// TwinCAT 3 PLC project Untitled1
// ProgramVersion: 3.1.4023.0
// libraries:
//   Tc2_MC2, * (Beckhoff Automation GmbH)
//   Tc2_Standard, * (Beckhoff Automation GmbH)
//   Tc2_System, * (Beckhoff Automation GmbH)
//   Tc2_Utilities, * (Beckhoff Automation GmbH)
//   Tc3_JsonXml, * (Beckhoff Automation GmbH)
//   Tc3_Module, * (Beckhoff Automation GmbH)
// project tree:
//   DUTs/ Bundle.TcDUT (not stored), Interval.TcDUT (not stored), PositionMaterials.TcDUT, SuctionPad.TcDUT (not stored)
//   DUTs/Enums/ A22.TcDUT (not stored), Cardboard.TcDUT (not stored), CornerGuard.TcDUT (not stored), Homing.TcDUT (not stored), SectionEnum.TcDUT (not stored), Surface.TcDUT
//   DUTs/Insertion/Drives/ ClearLinkMC.TcPOU, ServoNC.TcPOU, SimplePiston.TcPOU (not stored), TeknicHW.TcPOU (not stored)
//   DUTs/Insertion/ Insertion.TcPOU (not stored)
//   DUTs/Insertion/ABSTRACT/ FBA_Drive.TcPOU (not stored), I_ContinuousDrive.TcIO (not stored), I_Drive.TcIO (not stored), I_EncodedDrive.TcIO (not stored), I_PositionalDrive.TcIO (not stored)
//   DUTs/Machines/ FoldingMachine.TcPOU (not stored), KukaRobot.TcPOU (not stored), RobotA22.TcPOU, WrapMachine.TcPOU (not stored)
//   DUTs/Material Holders/ MaterialHolder.TcPOU, SkidMagazine.TcPOU (not stored), HmiSlotOccupancy.TcDUT
//   GVLs/ ContainerArrays.TcGVL, GVL.TcGVL (not stored), Hardware.TcGVL
//   / PlcTask.TcTTO (not stored)
//   POUs/A22 - Cardboard-Corner Guard/AOIs/ AOI_LoadCornerGuard.TcPOU, AOI_LoadFlatCardboard.TcPOU
//   POUs/A22 - Cardboard-Corner Guard/ CardboardCornerGuardEx.TcPOU
//   POUs/Hardware Calls/ SuctionQualityPtrArr.TcPOU (not stored), SetSuctionsPtrArr.TcPOU (not stored), CallHardwareModules.TcPOU, SuctionQuality.TcPOU, SetSuctions.TcPOU (not stored), SetupHardware.TcPOU
//   POUs/ MAIN.TcPOU, BundleJsonDemo.TcPOU
//   POUs/Materials/ GetMaterialLength.TcPOU (not stored), GetMaterialLengthFromCode.TcPOU (not stored), GetPairMasterLength.TcPOU (not stored), GetPositionMasterLength.TcPOU (not stored), MatchesMaterialType.TcPOU (not stored)
//   POUs/Utility/ CEILING.TcPOU (not stored), IntegerBitAccess.TcPOU, IntegerToBoolArray.TcPOU, WithinTolerance.TcPOU (not stored)
// real-time tasks:
//   TASK PlcTask: cycle T#10ms, priority 20, ADS port 350
// I/O:
//   DEVICE Device 1 (TC3 EIP Scanner), AmsNetId 5.131.216.41.2.1
//     ClearLink // <INFO> 169.254.0.152, ClearLink (ProdCode: 1, Rev: 2.93, Mac: 24:15:10:b0:30:37) </INFO> <EDS> C:\TwinCAT\3.1\Config\Io\EtherNetIP\clearlink_2.92.eds </EDS>

// ---- DUTs/Enums/Surface.TcDUT
{attribute 'qualified_only'}
//{attribute 'strict'}
TYPE Surface :
(
	TOP,
	LEFT,
	RIGHT,
	BOTTOM,
	
	TOP_LEFT,
	TOP_RIGHT,
	BOTTOM_LEFT,
	BOTTOM_RIGHT,
	
	size
);
END_TYPE

// ---- DUTs/Material Holders/HmiSlotOccupancy.TcDUT
TYPE HmiSlotOccupancy :
STRUCT
	material : STRING;
	occupied : BOOL;
END_STRUCT
END_TYPE

// ---- DUTs/PositionMaterials.TcDUT
TYPE PositionMaterials :
STRUCT
	position : REAL; //:= GVL.nullPos; //default value is set to predefined constant if bundle needs less than 32 position material pairs
	
	top : STRING;
	right : STRING;
	left : STRING;
	//sides : STRING;
	bottom : STRING;
	
	topLeft : STRING;
	topLeftFold : USINT;
	
	topRight : STRING;
	topRightFold : USINT;
	
	bottomLeft : STRING;
	bottomLeftFold : USINT;
	
	bottomRight : STRING;
	bottomRightFold : USINT;

	wrapPoints : USINT;
	wrapRotations : USINT;
END_STRUCT
END_TYPE

// ---- GVLs/ContainerArrays.TcGVL
//{attribute 'qualified_only'}
VAR_GLOBAL //data arrays to be passed into material holder FBs - do not access directly
	
	skidSlotsA22Left, skidSlotsA22Right : ARRAY[1..Cardboard.size-1] OF STRING; //cardboard skid
	skidOccupancyA22Left, skidOccupancyA22Right : ARRAY[1...Cardboard.size-1] OF BOOL := [(Cardboard.size-1)(TRUE)];
	skidHmiA22Left, skidHmiA22Right : ARRAY[1...Cardboard.size-1] OF HmiSlotOccupancy;
	
	magazineSlotsA22Left, magazineSlotsA22Right : ARRAY[1..CornerGuard.size-1] OF STRING; //corner guard magazine
	magazineOccupancyA22Left, magazineOccupancyA22Right : ARRAY[1..CornerGuard.size-1] OF BOOL := [(CornerGuard.size-1)(TRUE)];
	magazineHmiA22Left, magazineHmiA22Right : ARRAY[1..CornerGuard.size-1] OF HmiSlotOccupancy;
END_VAR

// ---- GVLs/Hardware.TcGVL
//{attribute 'qualified_only'}
VAR_GLOBAL //complete modules
	robot3, robot4 : RobotA22;
	
	benderA22Left : FoldingMachine;
	
	skidA22Left, skidA22Right : SkidMagazine;
	magazineA22Left, magazineA22Right : SkidMagazine;
	
	wrapperA22 : WrapMachine;
	overhead : STRING;
	
	horizontalDriveA22Left, horizontalDriveA22Right : ServoNC;
	verticalDriveA22Left, verticalDriveA22Right : ClearLinkMC;
	pistonA22Bottom : SimplePiston;
	
	(*
	each of these suction arrays are composed of 3 pads
	pad [2] is the corner pad used for corner guards
	pads [1] and [3] are the outer pads used for corner cardboards
	*)
	suctionA22TopLeft : ARRAY[1..3] OF SuctionPad;
	suctionA22TopRight : ARRAY[1..3] OF SuctionPad;
	suctionA22BottomLeft : ARRAY[1..3] OF SuctionPad; 
	suctionA22BottomRight : ARRAY[1..3] OF SuctionPad;
	
	suctionA22Bottom : SuctionPad;
END_VAR

// ---- DUTs/Machines/RobotA22.TcPOU
FUNCTION_BLOCK RobotA22 EXTENDS KukaRobot
VAR_OUTPUT //from outputs array
	taskID : A22;
	param1 : INT;
	param2 : INT;
	Xmm : INT;
	Ymm : INT;
	Zmm : INT;
	angle : INT;
	foldPosition0 : INT;
	foldPosition1 : INT;
END_VAR
VAR_OUTPUT //from inputs array
	tool : SectionEnum := SectionEnum.CARDBOARD_CORNERGUARD;
	suspendedMaterial : STRING;
	
	completedTask : A22;
	eoatDistance : INT;
	cardboardAvailability : INT;
	cornerGuardAvailability : INT;
	materialAtHoldingPosition : INT;
	//grp6
	//grp7
	
	wrapSafetyIn : BOOL;
	
END_VAR
VAR //HMI data
	reservationEnum : SectionEnum;
	hmiTask : STRING;
	hmiTool : STRING;
END_VAR

{warning disable C0195}
SUPER^();

outputs[1] := taskID;
outputs[2] := param1;
outputs[3] := param2;
outputs[4] := Xmm;
outputs[5] := Ymm;
outputs[6] := Zmm;
outputs[7] := angle;
outputs[8] := foldPosition0;
outputs[9] := foldPosition1;

refreshParameters();

reservationEnum := reservation;
IF reservationEnum = SectionEnum.NULL_SECTION THEN
	hmiReservation := 'N/A';
ELSE
	hmiReservation := TO_STRING(reservationEnum);
END_IF

hmiTask := TO_STRING(taskID);
hmiTool := TO_STRING(tool);

{attribute 'monitoring' := 'call'}
PROPERTY Busy : BOOL
GET
VAR
	//emptyOutput : ARRAY[1..50] OF INT;
END_VAR
//Busy stays TRUE until outputs are cleared AND completed task has elapsed
//Ready is always inverse of Busy
refreshParameters();

Busy := taskID <> 0 OR completedTask <> 0;
END_GET
END_PROPERTY

METHOD clearCommand : BOOL
VAR_INPUT
END_VAR
SUPER^.clearCommand();

refreshParameters();
END_METHOD

{attribute 'monitoring' := 'call'}
PROPERTY Done : BOOL
GET
refreshParameters();

Done :=
	completedTask = taskID AND
	taskID <> 0 AND
	completedTask <> 0;
END_GET
END_PROPERTY

{attribute 'monitoring' := 'call'}
PROPERTY HoldMaterial : STRING
GET
HoldMaterial := suspendedMaterial;
END_GET
SET
suspendedMaterial := HoldMaterial;
END_SET
END_PROPERTY

{attribute 'monitoring' := 'call'}
PROPERTY Ready : BOOL
GET
refreshParameters();

Ready := taskID = 0 AND completedTask = 0;
END_GET
END_PROPERTY

METHOD PRIVATE refreshParameters : BOOL
VAR_INPUT
END_VAR
{warning disable C0196}
taskID := outputs[1];
param1 := outputs[2];
param2 := outputs[3];
Xmm := outputs[4];
Ymm := outputs[5];
Zmm := outputs[6];
angle := outputs[7];
foldPosition0 := outputs[8];
foldPosition1 := outputs[9];

completedTask := inputs[1];
(*
eoatDistance := inputs[2];
magazineAvailability := inputs[3];
chipboardSkidInPosition := inputs[4];
materialAtHoldingPosition := inputs[5];
//robotEOAT := inputs[6];

strapSafetyIn := inputs[4].15;
*)
END_METHOD

METHOD setGroup : BOOL
VAR_INPUT
	group : INT;
	value : INT;
END_VAR
SUPER^.setGroup(group := group, value := value);

refreshParameters();
END_METHOD

METHOD setParameters : BOOL
VAR_INPUT
	newTaskID : INT;
	newParam1 : INT;
	newParam2 : INT;
	newXmm : INT;
	newYmm : INT;
	newZmm : INT;
	newAngle : INT;
	newStagingOccupancy : INT;
	newInsertionSuctionStatus : INT;
	newMagazineStatus : INT; //unused
	newInspectionValue : INT;
END_VAR
setGroup(group := 1, value := newTaskID);
setGroup(group := 2, value := newParam1);
setGroup(group := 3, value := newParam2);
setGroup(group := 4, value := newXmm);
setGroup(group := 5, value := newYmm);
setGroup(group := 6, value := newZmm);
setGroup(group := 7, value := newAngle);

newStagingOccupancy.15 := NOT wrapperA22.enable AND NOT wrapperA22.execute;
setGroup(group := 8, value := newStagingOccupancy);

setGroup(group := 9, value := newInsertionSuctionStatus);
setGroup(group := 10, value := newMagazineStatus);
setGroup(group := 11, value := newInspectionValue);

refreshParameters();
END_METHOD

END_FUNCTION_BLOCK

// ---- DUTs/Insertion/Drives/ServoNC.TcPOU
FUNCTION_BLOCK ServoNC EXTENDS FBA_Drive IMPLEMENTS I_EncodedDrive
VAR_OUTPUT	
	ready : BOOL;
	position : LREAL;
END_VAR
VAR
	axis : AXIS_REF;
	
	mcReadPosition : MC_ReadActualPosition;
	mcReset : MC_Reset;
	
	mcPower : MC_Power;
	mcMoveAbsolute : MC_MoveAbsolute;
	mcMoveRelative : MC_MoveRelative;
	mcMoveVelocity : MC_MoveVelocity;
	
	mcSetPosition : MC_SetPosition;
	mcStop : MC_Stop;
END_VAR
VAR_STAT CONSTANT
	targetingVelocity : INT := 500;
	continuousVelocity : INT := 200;
END_VAR

IF home OR outerLimit OR innerLimit THEN
	stop();
END_IF

blocks();

mcReset.Execute := FALSE;
mcMoveAbsolute.Execute := FALSE;
mcMoveRelative.Execute := FALSE;
mcMoveVelocity.Execute := FALSE;
mcSetPosition.Execute := FALSE;
mcStop.Execute := FALSE;

blocks();

ready := bEnable AND NOT busy AND homeSet;

METHOD PRIVATE blocks : BOOL
mcReadPosition(
	Axis:= axis, 
	Enable:= TRUE, 
	Valid=> , 
	Busy=> , 
	Error=> , 
	ErrorID=> , 
	Position=> position);

mcReset(
	Axis:= axis, 
	Execute:= , 
	Done=> , 
	Busy=> , 
	Error=> , 
	ErrorID=> );

mcPower(
	Axis:= axis, 
	Enable:= bEnable, 
	Enable_Positive:= TRUE, 
	Enable_Negative:= TRUE, 
	Override:= 100, 
	BufferMode:= , 
	Options:= , 
	Status=> , 
	Busy=> , 
	Active=> , 
	Error=> , 
	ErrorID=> );

mcMoveAbsolute(
	Axis:= axis, 
	Execute:= , 
	Position:= , 
	Velocity:= targetingVelocity, 
	Acceleration:= , 
	Deceleration:= , 
	Jerk:= , 
	BufferMode:= , 
	Options:= , 
	Done=> , 
	Busy=> , 
	Active=> , 
	CommandAborted=> , 
	Error=> , 
	ErrorID=> );
	
mcMoveRelative(
	Axis:= axis, 
	Execute:= , 
	Distance:= ,
	Velocity:= targetingVelocity, 
	Acceleration:= , 
	Deceleration:= , 
	Jerk:= , 
	BufferMode:= , 
	Options:= , 
	Done=> , 
	Busy=> , 
	Active=> , 
	CommandAborted=> , 
	Error=> , 
	ErrorID=> );
	
mcMoveVelocity( //stopped with stop();
	Axis:= axis, 
	Execute:= , 
	Velocity:= continuousVelocity, 
	Acceleration:= , 
	Deceleration:= , 
	Jerk:= , 
	Direction:= , 
	BufferMode:= , 
	Options:= , 
	InVelocity=> , 
	Busy=> , 
	Active=> , 
	CommandAborted=> , 
	Error=> , 
	ErrorID=> );
	
mcSetPosition(
	Axis:= axis, 
	Execute:= , 
	Position:= , 
	Mode:= , 
	Options:= , 
	Done=> , 
	Busy=> , 
	Error=> , 
	ErrorID=> );
	
mcStop(
	Axis:= axis, 
	Execute:= , 
	Deceleration:= , 
	Jerk:= , 
	Options:= , 
	Done=> , 
	Busy=> , 
	Active=> , 
	CommandAborted=> , 
	Error=> , 
	ErrorID=> );
END_METHOD

PROPERTY Busy : BOOL
GET
busy := 
	mcMoveAbsolute.Busy OR 
	mcMoveRelative.Busy OR 
	mcMoveVelocity.Busy OR 
	mcSetPosition.Busy OR 
	mcReset.Busy OR 
	mcStop.Busy OR 
	step <> 0;
END_GET
END_PROPERTY

PROPERTY CurrentPosition : LREAL
GET
CurrentPosition := position;
END_GET
SET
position := CurrentPosition;
END_SET
END_PROPERTY

PROPERTY Error : BOOL
GET
error := 
	mcMoveAbsolute.Error OR 
	mcMoveRelative.Error OR 
	mcMoveVelocity.Error OR 
	mcSetPosition.Error OR 
	mcReset.Error OR 
	mcStop.Error;
END_GET
END_PROPERTY

METHOD homingSequence : BOOL
CASE step OF
	Homing.IDLE:
		IF bEnable THEN
			step := Homing.IN;
		END_IF
		
	Homing.IN:
		IF mcMoveVelocity.Execute AND NOT innerLimit THEN
			mcMoveVelocity.Execute := FALSE;
			step := Homing.OUT;
			RETURN;
		END_IF
		
		mcMoveVelocity.Direction := MC_Negative_Direction;
		mcMoveVelocity.Execute := TRUE;
		
	Homing.OUT:
		IF mcMoveVelocity.Execute AND NOT home THEN //if reached home
			mcMoveVelocity.Execute := FALSE;
			step := Homing.STOP;
			RETURN;
		END_IF
		
		mcMoveVelocity.Direction := MC_Positive_Direction;
		mcMoveVelocity.Execute := TRUE;
		
	Homing.STOP:
		IF mcStop.Execute AND mcStop.Done THEN
			mcStop.Execute := FALSE;
			step := Homing.SET;
			RETURN;
		END_IF
		
		mcStop.Execute := TRUE;
		
	Homing.SET:
		IF mcSetPosition.Execute AND mcSetPosition.Done THEN
			mcSetPosition.Execute := FALSE;
			homingSequence := TRUE;
			step := Homing.IDLE;
			RETURN;
		END_IF
		
		mcSetPosition.Position := 0;
		mcSetPosition.Execute := TRUE;
		
END_CASE
END_METHOD

METHOD moveAbsolute : BOOL
VAR_INPUT
	newTarget : LREAL;
END_VAR
(*
VAR_OUTPUT
	fault : BOOL;
END_VAR
*)
IF NOT busy AND NOT error THEN
	mcMoveAbsolute.Position := newTarget;
	mcMoveAbsolute.Execute := TRUE;
END_IF

moveAbsolute := (*mcMoveAbsolute.Done AND mcMoveAbsolute.Active;*)
	position = newTarget;
END_METHOD

METHOD moveContinuous : BOOL
VAR_INPUT
	//direction : BOOL; //direction (F = inwards, T = outwards)
	direction : MC_Direction;
END_VAR
(*
IF mcMoveVelocity.Active THEN
	stop();
END_IF

IF NOT mcStop.Done THEN
	RETURN;
END_IF
*)
(*
IF direction THEN
	mcMoveVelocity.Direction := MC_Positive_Direction;
ELSE
	mcMoveVelocity.Direction := MC_Negative_Direction;
END_IF
*)
mcMoveVelocity.Direction := direction;

IF NOT mcMoveVelocity.Error THEN
	mcMoveVelocity.Execute := TRUE;
	moveContinuous := TRUE;
END_IF
END_METHOD

METHOD moveRelative : BOOL
VAR_INPUT
	distance : LREAL;
END_VAR
mcMoveRelative.Distance := distance;

moveRelative := mcMoveRelative.Done;
END_METHOD

METHOD reset : BOOL
VAR_INPUT
END_VAR
mcReset.Execute := TRUE;

reset := mcReset.Done;
END_METHOD

METHOD stop : BOOL
VAR_INPUT
END_VAR
mcStop.Execute := TRUE;
END_METHOD

PROPERTY TargetPosition : LREAL
GET
END_GET
SET
moveAbsolute(newTarget := TargetPosition);
END_SET
END_PROPERTY

END_FUNCTION_BLOCK

// ---- DUTs/Insertion/Drives/ClearLinkMC.TcPOU
FUNCTION_BLOCK ClearLinkMC EXTENDS FBA_Drive IMPLEMENTS I_EncodedDrive //I_PositionalDrive, I_ContinuousDrive
VAR_OUTPUT
	pulse AT %Q* : INT; //num pulses
	outputRegister AT %Q* : INT;
	brakeRelease AT %Q* : BOOL;
	
	A : BOOL; //direction (F = inwards, T = outwards)
	B : BOOL; //home bit
	clear : BOOL;
	
	hlfb AT %I* : REAL; //high level feedback, if -9999 then servo is idle
	position, targetPos : LREAL;
END_VAR
VAR
	pulseRequest : INT;
	
	minHoming : TON;
	resetTimer : TP;
	
	mode : (DISABLE, HOLD, TARGET, CONTINUOUS, RESET_ERR);
END_VAR
VAR_STAT CONSTANT
	resetTime : TIME := T#1000MS;
	unitsPerPulse : INT := 800; //800 Teknic units per revolution
	distancePerPulse : INT := 5; //5mm per revolution
END_VAR

//M-connector output register
outputRegister.0 := bEnable; 	//enable
outputRegister.1 := A; 			//direction bit
outputRegister.2 := B; 			//homing bit - set to TRUE after startup to begin homing, then set to FALSE to finish homing
outputRegister.3 := clear; 		//reset bit

resetTimer(IN:= , PT:= resetTime, Q=> clear, ET=> ); //reset timer

IF NOT bEnable THEN
	homingComplete := FALSE;
	mode := HOLD;
END_IF

override(); //if sensor limits are reached, this method blocks motion that would exceed the limits

CASE mode OF		
	HOLD: //hold current position, no motion
		pulse := 0;
		pulseRequest := 0;
	
	TARGET:	//target a given position
		IF WithinTolerance(position, targetPos, distancePerPulse) THEN
			pulseRequest := 0;
			mode := HOLD;
			
		ELSIF NOT Busy THEN
			A :=  position < targetPos;
			(*
			2 options to traverse to a target position:
				a)  send all pulses at once - single continuous motion but may exceed limits
				b)  1 pulse at a time - choppy but safer
			*)
			//pulseRequest := TO_INT(ABS(position - targetPos)/distancePerPulse);
			pulseRequest := 1;
			
		END_IF
		
	CONTINUOUS: //single pulses in the direction specified by moveContinuous()
		pulseRequest := 1;
		
	RESET_ERR: //reset pulse, servo may need to be rehomed aftewards
		pulse := 0;
		pulseRequest := 0;
		resetTimer.IN := TRUE;
		
		IF resetTimer.Q THEN
			resetTimer.IN := FALSE;
			mode := HOLD;
		END_IF
		
END_CASE

sequence();

PROPERTY Busy : BOOL
GET
Busy := hlfb <> -9999;
END_GET
END_PROPERTY

PROPERTY CurrentPosition : LREAL
GET
CurrentPosition := position;
END_GET
SET
position := CurrentPosition;
END_SET
END_PROPERTY

PROPERTY Error : BOOL
GET
END_GET
END_PROPERTY

METHOD homingSequence : BOOL
minHoming(IN:= , PT:= T#1S, Q=> , ET=> ); //IN and OUT should be held for at least 1 second - may be removed for deployment

IF NOT bEnable THEN //homing does not begin until software enable
	RETURN;
END_IF

CASE step OF
	Homing.IDLE:
		bEnable := FALSE;
		A := FALSE;
		B := FALSE;
		brakeRelease := TRUE;
		
		homingComplete := FALSE;
		step := Homing.IN;
		
	Homing.IN: //let insertion drop to inner limit before homing
		bEnable := FALSE;
		A := FALSE;
		B := FALSE;
		brakeRelease := TRUE;
		
		minHoming.IN := TRUE;
		
		IF NOT innerLimit AND minHoming.Q THEN
			minHoming.IN := FALSE;
			step := Homing.OUT;
		END_IF
	
	Homing.OUT:
		bEnable := TRUE;
		A := FALSE;
		B := TRUE;
		brakeRelease := TRUE;
		
		minHoming.IN := TRUE;
		
		IF NOT home AND minHoming.Q THEN
			minHoming.IN := FALSE;
			step := Homing.DONE;
		END_IF
		
	Homing.DONE:
		bEnable := TRUE;
		A := FALSE;
		B := FALSE;
		brakeRelease := TRUE;
			
		position := 0;
		
		homingComplete := TRUE;
		homingSequence := TRUE;
		
		mode := HOLD;
		step := Homing.IDLE;
	
END_CASE
END_METHOD

METHOD moveAbsolute : BOOL
VAR_INPUT
	newTarget : LREAL;
END_VAR
targetPos := newTarget;
mode := TARGET;
END_METHOD

METHOD moveContinuous : BOOL
VAR_INPUT
	direction : MC_Direction;
END_VAR
IF direction = MC_Negative_Direction THEN
	A := FALSE;
ELSIF direction = MC_Positive_Direction THEN
	A := TRUE;
END_IF

mode := CONTINUOUS;
END_METHOD

METHOD moveRelative : BOOL
VAR_INPUT
	distance : LREAL;
END_VAR
targetPos := targetPos + distance;

mode := TARGET;
END_METHOD

METHOD PRIVATE override : BOOL
VAR_INPUT
END_VAR
(*
IF (*NOT*) home THEN //block outwards motion
	position := 0;
	IF A THEN
		mode := HOLD;
	END_IF
	
ELSIF (*NOT*) outerLimit AND_THEN A THEN //block outwards motion
	mode := HOLD;

ELSIF (*NOT*) innerLimit AND_THEN NOT A THEN //block inwards motion
	mode := HOLD;
	
END_IF
*)


IF
	((*NOT*) home AND_THEN A) OR
	((*NOT*) outerLimit AND_THEN A) OR
	((*NOT*) innerLimit AND_THEN NOT A)
THEN
	mode := HOLD;
END_IF


IF (*NOT*) home THEN //block outwards motion
	position := 0;
END_IF
END_METHOD

METHOD reset : BOOL
VAR_INPUT
END_VAR
mode := RESET_ERR;
END_METHOD

METHOD PRIVATE sequence : BOOL
VAR_INPUT
END_VAR
IF Busy THEN //servo is active
	IF A THEN //positive direction
		position := position + (distancePerPulse * pulse);
	ELSE //negative direction
		position := position - (distancePerPulse * pulse);
	END_IF
	pulse := 0; //pulses already received, can be set to 0 so position change is not compounded

ELSIF pulse = 0 THEN //servo is not active
	pulse := pulseRequest;
	pulseRequest := 0; //remove this if not working as intended
	
END_IF
END_METHOD

METHOD stop : BOOL
VAR_INPUT
END_VAR
mode := HOLD;
END_METHOD

PROPERTY TargetPosition : LREAL
GET
END_GET
SET
targetPos := TargetPosition;
END_SET
END_PROPERTY

END_FUNCTION_BLOCK

// ---- DUTs/Material Holders/MaterialHolder.TcPOU
FUNCTION_BLOCK MaterialHolder
VAR_IN_OUT
	slots : ARRAY[*] OF STRING;
	occupied : ARRAY[*] OF BOOL;
	
	hmiTable : ARRAY[*] OF HmiSlotOccupancy;
END_VAR

IF hmiTable <> 0 THEN
	writeHmiTable();
END_IF

METHOD clear : BOOL
VAR_INPUT
END_VAR
MEMSET(ADR(slots), 0, SIZEOF(slots));
END_METHOD

METHOD findSlot : BOOL
VAR_INPUT
	materialID : STRING;
END_VAR
VAR_OUTPUT
	index : INT := 0;
END_VAR
VAR
	i : DINT;
END_VAR
IF materialID = '' THEN
	RETURN;
END_IF

FOR i:=LOWER_BOUND(slots, 1) TO UPPER_BOUND(slots, 1) BY 1 DO
	IF slots[i] = materialID THEN
		index := TO_INT(i);
		findSlot := TRUE;
		RETURN;
	END_IF
END_FOR
END_METHOD

METHOD getSlot : STRING
VAR_INPUT
	i : DINT;
END_VAR
VAR_OUTPUT
	error : BOOL;
END_VAR
error := i < LOWER_BOUND(slots, 1) OR i > UPPER_BOUND(slots, 1);

IF error THEN
	RETURN;
END_IF

getSlot := slots[i];
END_METHOD

METHOD getSlotsAsArray : POINTER TO STRING
getSlotsAsArray := ADR(slots);
END_METHOD

METHOD isOccupied : BOOL
VAR_INPUT
	i : DINT;
END_VAR
VAR_OUTPUT
	errorBounds : BOOL;
END_VAR
errorBounds := i < LOWER_BOUND(slots, 1) OR i > UPPER_BOUND(slots, 1);

IF errorBounds THEN
	RETURN;
END_IF

isOccupied := occupied[i];
END_METHOD

METHOD setSlot : BOOL
VAR_INPUT
	i : INT;
	material : STRING;
END_VAR
VAR_OUTPUT
	error : BOOL;
END_VAR
IF i < LOWER_BOUND(slots, 1) OR i > UPPER_BOUND(slots, 1) THEN
	error := TRUE;
	RETURN;
END_IF

slots[i] := material;

IF hmiTable <> 0 THEN
	writeHmiTable();
END_IF
END_METHOD

METHOD PRIVATE writeHmiTable : BOOL
VAR
	i : DINT;
END_VAR
FOR i:=LOWER_BOUND(hmiTable, 1) TO UPPER_BOUND(hmiTable, 1) BY 1 DO
	hmiTable[i].material := slots[i];
	hmiTable[i].occupied := occupied[i];
END_FOR
END_METHOD

END_FUNCTION_BLOCK

// ---- POUs/A22 - Cardboard-Corner Guard/AOIs/AOI_LoadCornerGuard.TcPOU
FUNCTION_BLOCK AOI_LoadCornerGuard
VAR_INPUT
	execute : BOOL;
END_VAR
VAR_IN_OUT CONSTANT
	sectionID : SectionEnum;
END_VAR
VAR_IN_OUT
	robot : RobotA22;
	magazine : SkidMagazine;
	loadedMaterials : ARRAY[*] OF STRING;
END_VAR
VAR_INPUT
	surfaceID : Surface;
	material : STRING;
	
	suctions : POINTER TO SuctionPad; //access from 0 to numPads-1, not LOWER_BOUND to UPPER_BOUND
	numPads : DINT;
END_VAR
VAR_OUTPUT
	donePulse : BOOL; //this signal turns on 1 cycle after done turns true, should not affect the program structure
	done : BOOL;
	busy : BOOL;
	error : BOOL;
	
	recovery : BOOL;
	failCounter : INT;
END_VAR
VAR
	run : BOOL;
	trigger : R_TRIG;
	doneTrigger : R_TRIG;
	
	slot : INT;
	
	suctionTimer : TON;
	step : (IDLE, PREP_ROBOT, GET_FROM_STORAGE, LOAD_TO_INSERTION, COMPLETE, RECOVERY_IDLE, RECOVERY_REMOVE, RECOVERY_LOAD);
	
	i : DINT;
END_VAR
VAR CONSTANT
	suctionDelay : TIME := T#2S;
	suctionDistance : INT := 10;
END_VAR

{warning disable C0371}

trigger(CLK:= execute, Q=> );
doneTrigger(CLK:= done, Q=> donePulse);
busy := trigger.Q OR step > 0;

IF step > IDLE AND_THEN NOT preExecution() THEN //conditions to track before execution
	RETURN;
END_IF

(*
if required bunk was not found on table - restage entire table
if bunk was not loaded correctly - remove bunk, then restage entire table
*)
CASE step OF
	IDLE:
		IF trigger.Q THEN
			recovery := FALSE;
			done := FALSE;
			error := FALSE;
			step := PREP_ROBOT;
		END_IF
		
	PREP_ROBOT:
		robot.clearCommand();
		IF robot.Ready THEN
			step := GET_FROM_STORAGE;
			slot := 0;
		END_IF
		
	GET_FROM_STORAGE:		
		IF NOT magazine.findSlot(materialID := material, index => slot) THEN
			error := TRUE;
			RETURN;
		END_IF
		
		IF robot.eoatDistance < suctionDistance THEN //move from table to robot gripper
			robot.HoldMaterial := magazine.getSlot(i := slot, error => );
		END_IF
		
		IF robot.Done THEN
			step := COMPLETE;
			RETURN;
		ELSIF robot.materialAtHoldingPosition > 0 THEN
			step := LOAD_TO_INSERTION;
			RETURN;
		END_IF
		
		CASE surfaceID OF
			Surface.TOP_LEFT, Surface.TOP_RIGHT:			robot.setGroup(group := 1, value := A22.LOAD_CORNER_GUARD_UPPER);
			Surface.BOTTOM_LEFT, SURFACE.BOTTOM_RIGHT:		robot.setGroup(group := 1, value := A22.LOAD_CORNER_GUARD_LOWER);
		END_CASE
		robot.setGroup(group := 2, value := slot); 
			
	LOAD_TO_INSERTION:
		IF robot.materialAtHoldingPosition > 0 AND robot.HoldMaterial <> '' THEN //move from gripper to insertion
			loadedMaterials[surfaceID] := robot.HoldMaterial;
			robot.HoldMaterial := '';
		END_IF
		
		//numPads/3 <= i < numPads/3 * 2
		FOR i:=(numPads/3)*1 TO (numPads/3)*2-1 BY 1 DO //middle third suctions only
			suctions[i].enable := TRUE;
		END_FOR
		
		IF robot.Done THEN
			suctionTimer.IN := FALSE;
			step := COMPLETE;
			RETURN;
		END_IF
		
		suctionTimer(IN:= , PT:= suctionDelay, Q=> , ET=> );
		suctionTimer.IN := TRUE;
		
		IF suctionTimer.Q THEN
			robot.setGroup(group := 10, value := robot.materialAtHoldingPosition);
		END_IF
	
	COMPLETE:
		robot.clearCommand();
		
		IF //check insertion quality
			SuctionQualityPtrArr(
				suctions := suctions, 
				numPads := numPads, 
				insertionMaterial := loadedMaterials[surfaceID], 
				recipeMaterial := material)
		THEN
			done := TRUE;
			slot := 0;
			step := 0;
			
		ELSE //recovery - remove and reload
			failCounter := failCounter + 1;
			step := RECOVERY_IDLE;
		END_IF
		
		
	//---------RECOVERY-----------------------------------------
	RECOVERY_IDLE:
		robot.clearCommand();
		IF robot.Ready THEN
			step := RECOVERY_REMOVE;
		END_IF
		
	RECOVERY_REMOVE:
		IF robot.Done THEN
			step := RECOVERY_LOAD;
			RETURN;
		END_IF
		
		CASE surfaceID OF
			Surface.TOP_LEFT, Surface.TOP_RIGHT:			robot.setGroup(group := 1, value := A22.REMOVE_CORNER_GUARD_UPPER);
			Surface.BOTTOM_LEFT, SURFACE.BOTTOM_RIGHT:		robot.setGroup(group := 1, value := A22.REMOVE_CORNER_GUARD_LOWER);
		END_CASE
		
	RECOVERY_LOAD:	
		recovery := TRUE;
		error := TRUE;
		
END_CASE

METHOD PRIVATE preExecution : BOOL
VAR_INPUT
END_VAR
{warning disable C0371}
IF material = '' THEN
	done := TRUE;
	RETURN;
END_IF

IF //robot must be ready before execution
	robot.error OR 
	robot.reservation <> sectionID OR 
	robot.tool <> sectionID
THEN
	error := TRUE;
	RETURN;
END_IF

preExecution := TRUE;
END_METHOD

METHOD reset : BOOL
VAR_INPUT
END_VAR
done := FALSE;
error := FALSE;
recovery := FALSE;
slot := 0;
step := 0;

failCounter := 0;
END_METHOD

END_FUNCTION_BLOCK

// ---- POUs/A22 - Cardboard-Corner Guard/AOIs/AOI_LoadFlatCardboard.TcPOU
FUNCTION_BLOCK AOI_LoadFlatCardboard
VAR_INPUT
	execute : BOOL;
END_VAR
VAR_IN_OUT CONSTANT
	sectionID : SectionEnum;
END_VAR
VAR_IN_OUT
	robot : RobotA22;
	skid : SkidMagazine;
	loadedMaterials : ARRAY[*] OF STRING;
END_VAR
VAR_INPUT
	surfaceID : Surface;
	material : STRING;
	
	suctions : POINTER TO SuctionPad; //access from 0 to numPads-1, not LOWER_BOUND to UPPER_BOUND
	numPads : DINT;
END_VAR
VAR_OUTPUT
	donePulse : BOOL;
	done : BOOL;
	busy : BOOL;
	error : BOOL;
	
	recovery : BOOL;
	failCounter : INT;
END_VAR
VAR
	run : BOOL;
	trigger : R_TRIG;
	doneTrigger : R_TRIG;
	
	slot : INT;
	
	suctionTimer : TON;
	step : (IDLE, PREP_ROBOT, GET_FROM_STORAGE, LOAD_TO_INSERTION, COMPLETE, RECOVERY_IDLE, RECOVERY_REMOVE, RECOVERY_WAIT, RECOVERY_LOAD);
	
	i : DINT;
END_VAR
VAR_STAT CONSTANT
	suctionDelay : TIME := T#2S;
	suctionDistance : INT := 10;
END_VAR

{warning disable C0371}

trigger(CLK:= execute, Q=> );
doneTrigger(CLK:= done, Q=> donePulse);
busy := trigger.Q OR step > 0;

IF step > IDLE AND_THEN NOT preExecution() THEN //conditions to track before execution
	RETURN;
END_IF

(*
if bunk was not loaded correctly - remove bunk, then restage entire table
*)
CASE step OF
	IDLE:
		IF trigger.Q THEN
			recovery := FALSE;
			done := FALSE;
			error := FALSE;
			step := PREP_ROBOT;
		END_IF
		
	PREP_ROBOT:
		robot.clearCommand();
		IF robot.Ready THEN
			step := GET_FROM_STORAGE;
			slot := 0;
		END_IF
		
	GET_FROM_STORAGE:		
		IF NOT skid.findSlot(materialID := material, index => slot) THEN
			error := TRUE;
			RETURN;
		END_IF
		
		IF robot.eoatDistance < suctionDistance THEN//move from table to robot gripper
			robot.HoldMaterial := skid.getSlot(i := slot, error => );;
		END_IF
		
		IF robot.Done THEN
			step := COMPLETE;
			RETURN;
		ELSIF robot.materialAtHoldingPosition >= 1 AND robot.materialAtHoldingPosition <= 8 THEN
			step := LOAD_TO_INSERTION;
			RETURN;
		END_IF
		
		CASE surfaceID OF
			Surface.TOP_LEFT, Surface.TOP_RIGHT:			robot.setGroup(group := 1, value := A22.LOAD_CORNER_GUARD_UPPER);
			Surface.BOTTOM_LEFT, SURFACE.BOTTOM_RIGHT:		robot.setGroup(group := 1, value := A22.LOAD_CORNER_GUARD_LOWER);
		END_CASE
		robot.setGroup(group := 2, value := slot); 
			
	LOAD_TO_INSERTION:
		IF robot.materialAtHoldingPosition > 0 AND robot.HoldMaterial <> '' THEN //move from gripper to insertion
			loadedMaterials[surfaceID] := robot.HoldMaterial;
			robot.HoldMaterial := '';
		END_IF
		
		//only bottom cardboard uses suction
		CASE surfaceID OF
			Surface.BOTTOM:		SetSuctionsPtrArr(suctions := suctions, numPads := numPads, state := TRUE);
		END_CASE
		
		IF robot.Done THEN
			suctionTimer.IN := FALSE;
			step := COMPLETE;
			RETURN;
		END_IF
		
		suctionTimer(IN:= , PT:= suctionDelay, Q=> , ET=> );
		suctionTimer.IN := TRUE;
		
		IF suctionTimer.Q THEN
			robot.setGroup(group := 10, value := robot.materialAtHoldingPosition);
		END_IF
	
	COMPLETE:
		robot.clearCommand();
		
		IF //if bottom then check insertion, otherwise done
			surfaceID <> Surface.BOTTOM OR_ELSE 
			SuctionQualityPtrArr(
				suctions := suctions, 
				numPads := numPads, 
				insertionMaterial := loadedMaterials[surfaceID], 
				recipeMaterial := material)
		THEN
			done := TRUE;
			slot := 0;
			step := 0;
			
		ELSE //recovery - remove and reload
			failCounter := failCounter + 1;
			step := RECOVERY_IDLE;
		END_IF
		
	//---------RECOVERY-----------------------------------------
	RECOVERY_IDLE:
		robot.clearCommand();
		IF robot.Ready THEN
			step := RECOVERY_REMOVE;
		END_IF
		
	RECOVERY_REMOVE:
		IF robot.Done THEN
			step := RECOVERY_LOAD;
			RETURN;
		END_IF
		
		CASE surfaceID OF
			Surface.BOTTOM:		robot.setGroup(group := 1, value := A22.REMOVE_CARDBOARD_BOTTOM);
		END_CASE
		
	RECOVERY_LOAD:	
		recovery := TRUE;
		error := TRUE;
		
END_CASE

METHOD PRIVATE preExecution : BOOL
VAR_INPUT
END_VAR
{warning disable C0371}
IF material = '' THEN
	done := TRUE;
	RETURN;
END_IF

IF //robot must be ready before execution
	robot.error OR 
	robot.reservation <> sectionID OR 
	robot.tool <> sectionID
THEN
	error := TRUE;
	RETURN;
END_IF

preExecution := TRUE;
END_METHOD

METHOD reset : BOOL
VAR_INPUT
END_VAR
done := FALSE;
error := FALSE;
recovery := FALSE;
slot := 0;
step := 0;

failCounter := 0;
END_METHOD

END_FUNCTION_BLOCK

// ---- POUs/A22 - Cardboard-Corner Guard/CardboardCornerGuardEx.TcPOU
FUNCTION_BLOCK CardboardCornerGuardEx
VAR_IN_OUT //controls
	execute : BOOL;
	stop : BOOL;
	
	manualStep : BOOL;
	manualSuction : BOOL;
END_VAR
VAR_IN_OUT
	benderLeft : FoldingMachine;
	
	robotLeft, robotRight : RobotA22;
	
	skidLeft, skidRight : SkidMagazine;
	magazineLeft, magazineRight : SkidMagazine;
	
	wrapper : WrapMachine;
	
	horizontalDriveLeft, horizontalDriveRight : ServoNC;
	verticalDriveLeft, verticalDriveRight : ClearLinkMC;
	pistonBottom : SimplePiston;
	
	suctionTopLeft : ARRAY[*(*1..3*)] OF SuctionPad;
	suctionTopRight : ARRAY[*(*1..3*)] OF SuctionPad;
	suctionBottomLeft : ARRAY[*(*1..3*)] OF SuctionPad; 
	suctionBottomRight : ARRAY[*(*1..3*)] OF SuctionPad;
END_VAR
VAR_OUTPUT
	generalError : BOOL;
	failLeft, failRight : BOOL;
END_VAR
VAR //for testing only
	latchLeft, latchRight : BOOL; //prevents sliders from overshooting the inner limit sensor
	
	suctionEnableTopLeft : BOOL;
	suctionEnableTopRight : BOOL;
	suctionEnableBottomLeft : BOOL;
	suctionEnableBottomRight : BOOL;
	
	ready : BOOL;
	done : BOOL;
END_VAR
VAR	
	step : (IDLE, LOAD_CORNERS, LOAD_FLATS, PUSH, TARGET_WRAP_POSITION, WRAP_AND_RELEASE, COMPLETE := 1050);
	iPair : INT;
	
	masterLoadStep : INT;
	loadSet : INT;
	loadStepLeft, loadStepRight : INT;
	cornerSetLeft, cornerSetRight : INT;
	
	iWrap : INT;
	wrapPoints : INT;
	wrapRotations : INT;
	masterLength : INT;
	
	releaseDelayTimer : TON;
END_VAR
VAR //local types
	topLeftFoldsArr, topRightFoldsArr, bottomLeftFoldsArr, bottomRightFoldsArr : ARRAY[0..GVL.maxPairs] OF INT;
	materialsArr : ARRAY[0..GVL.maxPairs] OF PositionMaterials := [
		(
			position := 0,
			top := 'CAR20M',
			left := 'CAR20S',
			right := 'CAR20S',
			bottom := 'CAR20L',
			topLeft := 'CAR28M',
			topRight := 'CAR28S',
			bottomLeft := 'CAR28S',
			bottomRight := 'CAR28L',
			wrapPoints := 1,
			wrapRotations := 4
		),
		(
			position := 0,
			topLeft := 'COR48',
			topRight := 'COR48',
			bottomLeft := 'COR48',
			bottomRight := 'COR48'
		)];
	
	demoHeight : REAL := 600; //600mm, 60cm
	
	insertionLeft, insertionRight : Insertion;
	innerLoadedMaterials, outerLoadedMaterials : ARRAY[Surface.TOP..Surface.BOTTOM_RIGHT] OF STRING;
	//inner: cardboard by default
	//outer: corner guard by default
END_VAR
VAR CONSTANT
	sectionID : SectionEnum := SectionEnum.CARDBOARD_CORNERGUARD;
	releaseDelay : TIME := T#2000MS;
END_VAR
VAR
	//AOIs encapsulate functionality and reduce the number of module variables
	aoiLoadCornerGuardLeft, aoiLoadCornerGuardRight : AOI_LoadCornerGuard;
	aoiLoadFlatCardboardLeft, aoiLoadFlatCardboardRight : AOI_LoadFlatCardboard;
END_VAR

callLocalModules();

IF stop THEN //may need to turn off suction
	insertionLeft.stop();
	insertionRight.stop();
	pistonBottom.stop();
	
	robotLeft.clearCommand();
	robotRight.clearCommand();
	RETURN;
END_IF

IF NOT (insertionLeft.homingComplete AND insertionRight.homingComplete) THEN
	insertionLeft.homingSequence();
	insertionRight.homingSequence();
	pistonBottom.retract();
END_IF

CASE step OF
	IDLE:
		IF execute THEN
			execute := FALSE;
			step := LOAD_CORNERS;
		END_IF
	
	LOAD_CORNERS:
		IF load(pairIndex := iPair) THEN
			IF manualStep AND_THEN NOT execute THEN
				RETURN;
			END_IF
		
			step := LOAD_FLATS;
		END_IF

	LOAD_FLATS:
		IF loadFlats(pair := materialsArr[iPair]) THEN
			IF manualStep AND_THEN NOT execute THEN
				RETURN;
			END_IF
			
			step := PUSH;
		END_IF
		
	PUSH:
		IF
			NOT insertionLeft.align(1000-demoHeight) OR
			NOT insertionRight.align(1000-demoHeight)
		THEN
			RETURN;
		END_IF
		
		insertionLeft.press();
		insertionRight.press();
		pistonBottom.extend();
		
		IF pistonBottom.extended AND insertionLeft.contact AND insertionRight.contact THEN
			step := TARGET_WRAP_POSITION;
		END_IF
		
	TARGET_WRAP_POSITION:		
		IF iWrap >= wrapPoints THEN
			step := COMPLETE;
			RETURN;
		END_IF
		
		//loadNextPair := materialsArr[iPair].position = materialsArr[iPair + 1].position;	
		
		IF materialsArr[iPair].position = materialsArr[iPair + 1].position THEN
			masterLength := MAX( GetPairMasterLength(materialsArr[iPair]), GetPairMasterLength(materialsArr[iPair + 1]) );
			wrapPoints := MAX( materialsArr[iPair].wrapPoints, materialsArr[iPair + 1].wrapPoints );
			wrapRotations := MAX( materialsArr[iPair].wrapRotations, materialsArr[iPair + 1].wrapRotations );
		ELSE
			masterLength := GetPairMasterLength(materialsArr[iPair]);
			wrapPoints := materialsArr[iPair].wrapPoints;
			wrapRotations := materialsArr[iPair].wrapRotations;
		END_IF
		
		(*
		directionCheckAndSet(
			wrapConveyorPos,
			(currentPair.position - masterLength/2) + (masterLength/(currentPair.wrapPoints + 1) * (iWrap + 1)));
		*)
		step := WRAP_AND_RELEASE;
		
	WRAP_AND_RELEASE:
		releaseDelayTimer(IN:= , PT:= releaseDelay, Q=> , ET=> );
		
		IF wrapper.ready THEN
			wrapper.wrap(wrapRotations);
			releaseDelayTimer.IN := TRUE;
		END_IF
		
		IF releaseDelayTimer.Q THEN
			SetSuctions(suctions := suctionTopLeft, state := FALSE);
			SetSuctions(suctions := suctionTopRight, state := FALSE);
			SetSuctions(suctions := suctionBottomLeft, state := FALSE);
			SetSuctions(suctions := suctionBottomRight, state := FALSE);
			
			insertionLeft.align(0);
			insertionRight.align(0);
			insertionLeft.release();
			insertionRight.release();
			
			pistonBottom.retract();
		END_IF
		
		IF wrapper.done AND insertionLeft.home AND insertionRight.home AND pistonBottom.retracted THEN
			releaseDelayTimer.IN := FALSE;
			step := WRAP_AND_RELEASE;
		END_IF
	
	COMPLETE:
		iPair := (iPair + 1) MOD GVL.maxPairs;
		iWrap := wrapPoints := wrapRotations := 0;
		step := IDLE;
		
END_CASE

ACTION blocks:
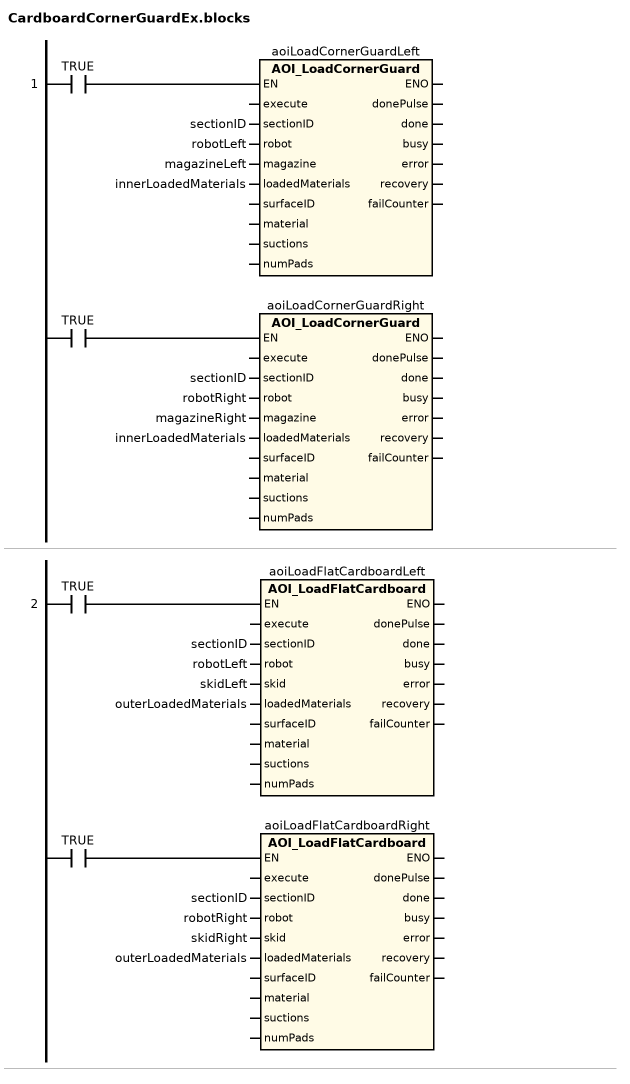
// NETWORK 1
aoiLoadCornerGuardLeft(
    sectionID := sectionID,
    robot := robotLeft,
    magazine := magazineLeft,
    loadedMaterials := innerLoadedMaterials); // AOI_LoadCornerGuard
aoiLoadCornerGuardRight(
    sectionID := sectionID,
    robot := robotRight,
    magazine := magazineRight,
    loadedMaterials := innerLoadedMaterials); // AOI_LoadCornerGuard

// NETWORK 2
aoiLoadFlatCardboardLeft(
    sectionID := sectionID,
    robot := robotLeft,
    skid := skidLeft,
    loadedMaterials := outerLoadedMaterials); // AOI_LoadFlatCardboard
aoiLoadFlatCardboardRight(
    sectionID := sectionID,
    robot := robotRight,
    skid := skidRight,
    loadedMaterials := outerLoadedMaterials); // AOI_LoadFlatCardboard
END_ACTION

ACTION callLocalModules:
{warning disable C0371}
insertionLeft(
	enable:= TRUE, 
	slider:= verticalDriveLeft, 
	screw:= horizontalDriveLeft, 
	contact=> , 
	softContact=> , 
	busy=> , 
	error=> , 
	home=> , 
	homingComplete=> , 
	sliderPos=> );
	
insertionRight(
	enable:= TRUE, 
	slider:= verticalDriveRight, 
	screw:= horizontalDriveRight, 
	contact=> , 
	softContact=> , 
	busy=> , 
	error=> , 
	home=> , 
	homingComplete=> , 
	sliderPos=> );
END_ACTION

METHOD PROTECTED leftCornerSequence : BOOL
VAR_IN_OUT
	robot : RobotA22;
	skid : SkidMagazine;
	suctions : POINTER TO SuctionPad; //ARRAY[*] OF SuctionPad;
	loadStep : INT;
END_VAR
VAR_INPUT
	surfaceID : Surface;
	material : STRING;
	foldPos0 : INT;
	foldPos1 : INT;
END_VAR
VAR_OUTPUT
	error : BOOL;
END_VAR
VAR
	column : INT;
END_VAR
VAR CONSTANT
	suctionDistance : INT := 10;
END_VAR
{warning disable C0371}
IF material = '' THEN
	leftCornerSequence := TRUE;
	RETURN;
END_IF

benderLeft.setFoldingPositions(foldPos0, foldPos1);

CASE loadStep OF
	0:
		robot.clearCommand();
		IF robot.Ready AND overhead = '' THEN
			loadStep := 10;
		END_IF
		
	10: //skid to bender
		IF NOT skid.findSlot(materialID:= material, index=> column) THEN
			error := TRUE;
			RETURN;
		END_IF
		
		(*
		IF robot.eoatDistance < suctionDistance THEN
			robot.HoldMaterial := skid.getSlot(i := column);
		END_IF
		*)
		
		IF robot.Done THEN
			loadStep := 20;
			RETURN;
		END_IF
		
		robot.setGroup(group := 1, value := A22.TRANSFER_TO_BENDER);
		robot.setGroup(group := 2, value := foldPos0);
		robot.setGroup(group := 3, value := foldPos1);
		
	20: //bend
		//IF benderLeft.done THEN
			loadStep := 30;
		//END_IF
		
	30: //bender to overhead or left insertion
		IF wrapper.trayOccupied AND wrapper.Overhead = '' AND robot.HoldMaterial <> '' THEN
			wrapper.Overhead := robot.HoldMaterial;
			robot.HoldMaterial := '';
		END_IF
	
		IF robot.Done THEN
			loadStep := COMPLETE;
			RETURN;
		END_IF
		
		CASE surfaceID OF
			Surface.TOP_RIGHT:		robot.setGroup(group := 1, value := A22.TRANSFER_TO_OVERHEAD);
			Surface.BOTTOM_RIGHT:	robot.setGroup(group := 1, value := A22.TRANSFER_TO_OVERHEAD);
			Surface.TOP_LEFT:		robot.setGroup(group := 1, value := A22.LOAD_BENDER_TO_UPPER_CORNER);
			Surface.BOTTOM_LEFT:	robot.setGroup(group := 1, value := A22.LOAD_BENDER_TO_LOWER_CORNER);
		END_CASE
		robot.setGroup(group := 2, value := 0);
		robot.setGroup(group := 3, value := 0);
	
	COMPLETE:
		CASE surfaceID OF
			Surface.TOP_LEFT:		suctionTopLeft[1].enable := suctionTopLeft[3].enable := TRUE;
			Surface.BOTTOM_LEFT:	suctionBottomLeft[1].enable := suctionBottomLeft[3].enable := TRUE;
		END_CASE
		
		leftCornerSequence := TRUE;
		
END_CASE
END_METHOD

METHOD PROTECTED load : BOOL
VAR_INPUT
	pairIndex : INT;
END_VAR
VAR
	pair : REFERENCE TO PositionMaterials REF= materialsArr[pairIndex];
	nextPair : REFERENCE TO PositionMaterials;
END_VAR
(*
unlike other sections, the load() function for cardboard + corner guard only loads the corners
to load flat cardboards, use the function loadFlats()
*)
{warning disable C0371}

IF robotLeft.error OR robotRight.error THEN
	RETURN;
ELSIF NOT (robotLeft.reserve(sectionID) AND robotRight.reserve(sectionID)) THEN //both robots must be reserved first
	RETURN;
END_IF

IF pairIndex + 1 < GVL.maxPairs THEN
	nextPair REF= materialsArr[pairIndex + 1];
END_IF

CASE masterLoadStep OF
	0: //next pair (which is to be placed over this pair) has the same position as this pair
		IF pairIndex + 1 >= GVL.maxPairs THEN //no next pair
			masterLoadStep := 10;
		ELSIF pair.position < nextPair.position THEN
			masterLoadStep := 10;
		ELSIF MatchesMaterialType(pair:= nextPair, materialType:= 'CAR') AND_THEN loadCornerCardboards(pairIndex:= pairIndex + 1) THEN
			masterLoadStep := 10;
		ELSIF MatchesMaterialType(pair:= nextPair, materialType:= 'COR') AND_THEN loadCornerGuards(pairIndex:= pairIndex + 1) THEN
			masterLoadStep := 10;
		END_IF
		
	10:
		IF
			MatchesMaterialType(pair:= pair, materialType:= 'CAR') AND_THEN loadCornerCardboardsEx(pairIndex:= iPair) OR_ELSE
			MatchesMaterialType(pair:= pair, materialType:= 'COR') AND_THEN loadCornerGuards(pairIndex:= iPair)
		THEN //is cardboard
			masterLoadStep := COMPLETE;
		END_IF
	
	COMPLETE:
		robotLeft.release(sectionID);
		robotRight.release(sectionID);
		
		masterLoadStep := 0;
		load := TRUE;
	
END_CASE
END_METHOD

METHOD PROTECTED loadCornerCardboards : BOOL
VAR_INPUT
	pairIndex : INT;
END_VAR
VAR
	leftSuctionArr, rightSuctionArr : POINTER TO SuctionPad;
	leftNextSet, rightNextSet : INT;
	leftMaterial, rightMaterial : STRING;
	leftFold, rightFold : INT;
	
	pair : REFERENCE TO PositionMaterials REF= materialsArr[pairIndex];
	topLeftFold : INT := topLeftFoldsArr[pairIndex];
	topRightFold : INT := topRightFoldsArr[pairIndex];
	bottomLeftFold : INT := bottomLeftFoldsArr[pairIndex];
	bottomRightFold : INT := bottomRightFoldsArr[pairIndex];
END_VAR
{warning disable C0371}
CASE cornerSetLeft OF
	0:
		leftNextSet := Surface.TOP_RIGHT;
		cornerSetLeft := 0;
		
	Surface.TOP_RIGHT: 
		leftNextSet := Surface.TOP_LEFT;
		leftSuctionArr := suctionTopRight;
		leftMaterial := pair.topRight;
		leftFold := topRightFold;
		
	Surface.TOP_LEFT: 
		leftNextSet := Surface.BOTTOM_RIGHT;
		leftSuctionArr := suctionTopLeft;
		leftMaterial := pair.topLeft;
		leftFold := topLeftFold;
		
	Surface.BOTTOM_RIGHT:
		leftNextSet := Surface.BOTTOM_LEFT;
		leftSuctionArr := suctionBottomRight;
		leftMaterial := pair.bottomRight;
		leftFold := bottomRightFold;
		
	Surface.BOTTOM_LEFT: 
		leftNextSet := COMPLETE;
		leftSuctionArr := suctionBottomLeft;
		leftMaterial := pair.bottomLeft;
		leftFold := bottomLeftFold;
END_CASE
IF
	(cornerSetLeft = 0 OR cornerSetLeft = COMPLETE) OR_ELSE
	leftCornerSequence(
		robot:= robotLeft, 
		skid:= skidLeft, 
		suctions := leftSuctionArr,
		loadStep:= loadStepLeft, 
		surfaceID:= cornerSetLeft,
		material:= pair.topRight, 
		foldPos0:= topRightFold, 
		foldPos1:= 0, 
		error=> )
THEN
	cornerSetLeft := leftNextSet;
	loadStepLeft := 0;
END_IF


CASE cornerSetRight OF
	0:
		cornerSetRight := Surface.TOP_RIGHT;
		rightSuctionArr := suctionTopRight;
		
	Surface.TOP_RIGHT:		
		rightNextSet := Surface.BOTTOM_RIGHT;
		rightSuctionArr := suctionTopRight;
		rightMaterial := pair.topRight;
		rightFold := topRightFold;
		
	Surface.BOTTOM_RIGHT: 
		rightNextSet := COMPLETE;
		rightSuctionArr := suctionBottomRight;
		rightMaterial := pair.bottomRight;
		rightFold := bottomRightFold;		
END_CASE
IF
	(cornerSetRight = 0 OR cornerSetRight = COMPLETE) OR_ELSE
	rightCornerSequence(
		robot:= robotRight, 
		skid:= skidRight, 
		suctions := rightSuctionArr,
		loadStep:= loadStepRight, 
		material:= pair.topRight, 
		surfaceID:= cornerSetRight,
		foldPos0:= pair.topRightFold, 
		foldPos1:= 0, 
		error=> )
THEN
	cornerSetRight := rightNextSet;
	loadStepRight := 0;
END_IF



IF cornerSetLeft = COMPLETE AND cornerSetRight = COMPLETE THEN
	loadCornerCardboards := TRUE;
	
	loadStepLeft := loadStepRight := 0;
	cornerSetLeft := cornerSetRight := 0;
END_IF
END_METHOD

METHOD PROTECTED loadCornerCardboardsEx : BOOL
VAR_INPUT
	pairIndex : INT;
END_VAR
VAR
	suctionsArrLeft, suctionsArrRight : POINTER TO SuctionPad;
	nextSetLeft, nextSetRight : INT;

	pair : REFERENCE TO PositionMaterials REF= materialsArr[pairIndex];
	topLeftFold : INT := topLeftFoldsArr[pairIndex];
	topRightFold : INT := topRightFoldsArr[pairIndex];
	bottomLeftFold : INT := bottomLeftFoldsArr[pairIndex];
	bottomRightFold : INT := bottomRightFoldsArr[pairIndex];
END_VAR
{warning disable C0371}
CASE cornerSetLeft OF
	0:
		cornerSetLeft := Surface.TOP_RIGHT;
		loadStepLeft := 0;
		
	Surface.TOP_RIGHT: 
		IF
			leftCornerSequence(
				robot:= robotLeft, 
				skid:= skidLeft, 
				suctions := suctionTopRight,
				loadStep:= loadStepLeft, 
				surfaceID:= Surface.TOP_RIGHT,
				material:= pair.topRight, 
				foldPos0:= topRightFold, 
				foldPos1:= 0, 
				error=> )
		THEN
			cornerSetLeft := Surface.TOP_LEFT;
			loadStepLeft := 0;
		END_IF
		
	Surface.TOP_LEFT: 
		IF
			leftCornerSequence(
				robot:= robotLeft, 
				skid:= skidLeft, 
				suctions := suctionTopLeft,
				loadStep:= loadStepLeft, 
				surfaceID:= Surface.TOP_LEFT,
				material:= pair.topLeft, 
				foldPos0:= topLeftFold, 
				foldPos1:= 0, 
				error=> )
		THEN
			cornerSetLeft := Surface.BOTTOM_RIGHT;
			loadStepLeft := 0;
		END_IF
		
	Surface.BOTTOM_RIGHT: 
		IF
			leftCornerSequence(
				robot:= robotLeft, 
				skid:= skidLeft, 
				suctions := suctionBottomRight,
				loadStep:= loadStepLeft, 
				surfaceID:= Surface.BOTTOM_RIGHT,
				material:= pair.bottomRight, 
				foldPos0:= bottomRightFold, 
				foldPos1:= 0, 
				error=> )
		THEN
			cornerSetLeft := Surface.BOTTOM_LEFT;
			loadStepLeft := 0;
		END_IF
		
	Surface.BOTTOM_LEFT: 
		IF
			leftCornerSequence(
				robot:= robotLeft, 
				skid:= skidLeft, 
				suctions := suctionBottomLeft,
				loadStep:= loadStepLeft, 
				surfaceID:= Surface.BOTTOM_LEFT,
				material:= pair.bottomLeft, 
				foldPos0:= bottomLeftFold, 
				foldPos1:= 0, 
				error=> )
		THEN
			cornerSetLeft := COMPLETE;
			loadStepLeft := 0;
		END_IF
END_CASE

//------------------------------------------------------------
CASE cornerSetRight OF
	0:
		cornerSetRight := Surface.TOP_RIGHT;
		loadStepRight := 0;
		
	Surface.TOP_RIGHT: 
		IF
			rightCornerSequence(
				robot:= robotRight, 
				skid:= skidRight, 
				suctions := suctionTopRight,
				loadStep:= loadStepRight, 
				surfaceID:= Surface.TOP_RIGHT,
				material:= pair.topRight, 
				foldPos0:= topRightFold, 
				foldPos1:= 0, 
				error=> )
		THEN
			cornerSetRight := Surface.BOTTOM_RIGHT;
			loadStepRight := 0;
		END_IF
		
	Surface.BOTTOM_RIGHT: 
		IF
			rightCornerSequence(
				robot:= robotRight, 
				skid:= skidRight, 
				suctions := suctionBottomRight,
				loadStep:= loadStepRight, 
				surfaceID:= Surface.BOTTOM_RIGHT,
				material:= pair.bottomRight, 
				foldPos0:= bottomRightFold, 
				foldPos1:= 0, 
				error=> )
		THEN
			cornerSetRight := Surface.BOTTOM_RIGHT;
			loadStepRight := 0;
		END_IF
		
		cornerSetRight := COMPLETE;			
		loadStepRight := COMPLETE;
		
END_CASE

//------------------------------------------------------------
IF cornerSetLeft = COMPLETE AND cornerSetRight = COMPLETE THEN
	loadCornerCardboardsEx := TRUE;
	
	loadStepLeft := loadStepRight := 0;
	cornerSetLeft := cornerSetRight := 0;
END_IF
END_METHOD

METHOD PROTECTED loadCornerGuards : BOOL
VAR_INPUT
	pairIndex : INT;
END_VAR
VAR_OUTPUT
	fail : BOOL;
END_VAR
VAR
	pair : REFERENCE TO PositionMaterials REF= materialsArr[pairIndex];
END_VAR
{warning disable C0371}
CASE loadSet OF
	0: //upper corners
		IF 
			loadGuardSequence(
				robot:= robotLeft, 
				magazine:= magazineLeft, 
				suctions:= suctionTopLeft,
				loadStep:= loadStepLeft, 
				surfaceID:= Surface.TOP_LEFT, 
				material:= pair.topLeft, 
				error=> failLeft)
			AND
			loadGuardSequence(
				robot:= robotRight, 
				magazine:= magazineLeft,
				suctions:= suctionTopRight,
				loadStep:= loadStepRight, 
				surfaceID:= Surface.TOP_RIGHT, 
				material:= pair.topRight, 
				error=> failRight)
		THEN
			loadStepLeft := loadStepRight := 0;
			loadSet := 10;
		END_IF
		
	10: //lower corners
		IF 
			loadGuardSequence(
				robot:= robotLeft, 
				magazine:= skidLeft, 
				suctions:= suctionTopLeft,
				loadStep:= loadStepLeft, 
				surfaceID:= Surface.BOTTOM_LEFT, 
				material:= pair.bottomLeft, 
				error=> failLeft)
			AND
			loadGuardSequence(
				robot:= robotRight, 
				magazine:= skidRight,
				suctions:= suctionTopRight,
				loadStep:= loadStepRight, 
				surfaceID:= Surface.BOTTOM_RIGHT, 
				material:= pair.bottomRight, 
				error=> failRight)
		THEN
			loadStepLeft := loadStepRight := 0;
			loadSet := COMPLETE;
		END_IF
	
	COMPLETE:
		loadStepLeft := loadStepRight := 0;
		loadSet := 0;
		
		loadCornerGuards := TRUE;
END_CASE

fail := failLeft OR failRight;
END_METHOD

METHOD PROTECTED loadFlats : BOOL
VAR_INPUT
	pair : REFERENCE TO PositionMaterials;
END_VAR
VAR_OUTPUT
	error : BOOL;
END_VAR
{warning disable C0371}
CASE loadSet OF
	0: //top and bottom
		IF 
			loadFlatSequence(
				robot:= robotLeft, 
				skid:= skidLeft, 
				loadStep:= loadStepLeft, 
				surfaceID:= Surface.TOP, 
				material:= pair.top, 
				fail=> )
			AND
			loadFlatSequence(
				robot:= robotRight, 
				skid:= skidRight, 
				loadStep:= loadStepRight, 
				surfaceID:= Surface.BOTTOM, 
				material:= pair.bottom, 
				fail=> )
		THEN
			loadStepLeft := loadStepRight := 0;
			loadSet := 10;
		END_IF
		
	10: //sides
		IF 
			loadFlatSequence(
				robot:= robotLeft, 
				skid:= skidLeft, 
				loadStep:= loadStepLeft, 
				surfaceID:= Surface.LEFT, 
				material:= pair.left, 
				fail=> )
			AND
			loadFlatSequence(
				robot:= robotRight, 
				skid:= skidRight, 
				loadStep:= loadStepRight, 
				surfaceID:= Surface.RIGHT, 
				material:= pair.right, 
				fail=> )
		THEN
			loadStepLeft := loadStepRight := 0;
			loadSet := COMPLETE;
		END_IF
	
	COMPLETE:
		loadStepLeft := loadStepRight := 0;
		loadSet := 0;
		
		loadFlats := TRUE;
END_CASE
END_METHOD

METHOD loadFlatSequence : BOOL
VAR_IN_OUT
	robot : RobotA22;
	skid : SkidMagazine;
	loadStep : INT;
END_VAR
VAR_INPUT
	surfaceID : Surface;
	material : STRING;
END_VAR
VAR_OUTPUT
	fail : BOOL;
END_VAR
VAR
	task : INT;
	slot : INT;
END_VAR
IF material = '' THEN
	loadFlatSequence := TRUE;
	RETURN;
END_IF

CASE loadStep OF
	0:
		robot.clearCommand();
		IF robot.Ready THEN
			step := 10;
		END_IF
		
	10: //storage to gripper
		IF NOT skid.findSlot(materialID := material, index => slot) THEN
			fail := TRUE;
			RETURN;
		END_IF
		
		IF robot.Done THEN
			loadStep := COMPLETE;
			RETURN;
		END_IF
		
		CASE surfaceID OF
			Surface.TOP: 					task := A22.LOAD_CARDBOARD_TOP;
			Surface.LEFT, Surface.RIGHT: 	task := A22.LOAD_CARDBOARD_SIDE;
			Surface.BOTTOM: 				task := A22.LOAD_CARDBOARD_BOTTOM;
		END_CASE
		
		robot.setGroup(group := 1, value := task);
		robot.setGroup(group := 2, value := slot);
		
	20: //gripper to insertion
		
	COMPLETE:
		loadFlatSequence := TRUE;
	
END_CASE
END_METHOD

METHOD loadGuardSequence : BOOL
VAR_IN_OUT
	robot : RobotA22;
	magazine : SkidMagazine;
	suctions : ARRAY[*] OF SuctionPad;
	loadStep : INT;
END_VAR
VAR_INPUT
	surfaceID : Surface;
	material : STRING;
END_VAR
VAR_OUTPUT
	error : BOOL;
END_VAR
VAR
	task : INT;
	slot : INT;
END_VAR
IF material = '' THEN
	loadGuardSequence := TRUE;
	RETURN;
END_IF

CASE loadStep OF
	0:
		IF NOT magazine.findSlot(materialID := material, index => slot) THEN //load from staging table
			error := TRUE;
			RETURN;
		END_IF
		
		IF robot.Done THEN
			loadStep := COMPLETE;
			RETURN;
		END_IF
		
		CASE surfaceID OF
			Surface.TOP_LEFT, Surface.TOP_RIGHT: 		task := A22.LOAD_CORNER_GUARD_UPPER;
			Surface.BOTTOM_LEFT, Surface.BOTTOM_RIGHT:	task := A22.LOAD_CORNER_GUARD_LOWER;
		END_CASE
		
		robot.setGroup(group := 1, value := task);
		robot.setGroup(group := 2, value := slot);
		
	COMPLETE:
		suctions[2].enable := TRUE;
		loadGuardSequence := TRUE;
END_CASE
END_METHOD

METHOD PROTECTED loadLeftCornerCardboards : BOOL
VAR_INPUT
	pair : REFERENCE TO PositionMaterials;
END_VAR
VAR
	suctionsArrLeft, suctionsArrRight : POINTER TO SuctionPad;
	nextSetLeft, nextSetRight : INT;
END_VAR
{warning disable C0371}
CASE cornerSetLeft OF
	0:
		cornerSetLeft := Surface.TOP_RIGHT;
		loadStepLeft := 0;
		
	Surface.TOP_RIGHT: 
		IF
			leftCornerSequence(
				robot:= robotLeft, 
				skid:= skidLeft, 
				suctions := suctionTopRight,
				loadStep:= loadStepLeft, 
				surfaceID:= Surface.TOP_RIGHT,
				material:= pair.topRight, 
				foldPos0:= pair.topRightFold, 
				foldPos1:= 0, 
				error=> )
		THEN
			cornerSetLeft := Surface.TOP_LEFT;
			loadStepLeft := 0;
		END_IF
		
	Surface.TOP_LEFT: 
		IF
			leftCornerSequence(
				robot:= robotLeft, 
				skid:= skidLeft, 
				suctions := suctionTopLeft,
				loadStep:= loadStepLeft, 
				surfaceID:= Surface.TOP_LEFT,
				material:= pair.topLeft, 
				foldPos0:= pair.topLeftFold, 
				foldPos1:= 0, 
				error=> )
		THEN
			cornerSetLeft := Surface.BOTTOM_RIGHT;
			loadStepLeft := 0;
		END_IF
		
	Surface.BOTTOM_RIGHT: 
		IF
			leftCornerSequence(
				robot:= robotLeft, 
				skid:= skidLeft, 
				suctions := suctionBottomRight,
				loadStep:= loadStepLeft, 
				surfaceID:= Surface.BOTTOM_RIGHT,
				material:= pair.bottomRight, 
				foldPos0:= pair.bottomRightFold, 
				foldPos1:= 0, 
				error=> )
		THEN
			cornerSetLeft := Surface.BOTTOM_LEFT;
			loadStepLeft := 0;
		END_IF
		
	Surface.BOTTOM_LEFT: 
		IF
			leftCornerSequence(
				robot:= robotLeft, 
				skid:= skidLeft, 
				suctions := suctionBottomLeft,
				loadStep:= loadStepLeft, 
				surfaceID:= Surface.BOTTOM_LEFT,
				material:= pair.bottomLeft, 
				foldPos0:= pair.bottomLeftFold, 
				foldPos1:= 0, 
				error=> )
		THEN
			cornerSetLeft := COMPLETE;
			loadStepLeft := 0;
		END_IF
END_CASE

//------------------------------------------------------------
IF cornerSetLeft = COMPLETE THEN
	loadStepLeft := 0;
	cornerSetLeft := 0;
	loadLeftCornerCardboards := TRUE;
END_IF
END_METHOD

METHOD PROTECTED loadRightCornerCardboards : BOOL
VAR_INPUT
	pair : REFERENCE TO PositionMaterials;
END_VAR
VAR
	suctionsArrLeft, suctionsArrRight : POINTER TO SuctionPad;
	nextSetLeft, nextSetRight : INT;
END_VAR
{warning disable C0371}
CASE cornerSetRight OF
	0:
		cornerSetRight := Surface.TOP_RIGHT;
		loadStepRight := 0;
		
	Surface.TOP_RIGHT: 
		IF
			rightCornerSequence(
				robot:= robotRight, 
				skid:= skidRight, 
				suctions := suctionTopRight,
				loadStep:= loadStepRight, 
				surfaceID:= Surface.TOP_RIGHT,
				material:= pair.topRight, 
				foldPos0:= pair.topRightFold, 
				foldPos1:= 0, 
				error=> )
		THEN
			cornerSetRight := Surface.BOTTOM_RIGHT;
			loadStepRight := 0;
		END_IF
		
	Surface.BOTTOM_RIGHT: 
		IF
			rightCornerSequence(
				robot:= robotRight, 
				skid:= skidRight, 
				suctions := suctionBottomRight,
				loadStep:= loadStepRight, 
				surfaceID:= Surface.BOTTOM_RIGHT,
				material:= pair.bottomRight, 
				foldPos0:= pair.bottomRightFold, 
				foldPos1:= 0, 
				error=> )
		THEN
			cornerSetRight := Surface.BOTTOM_RIGHT;
			loadStepRight := 0;
		END_IF
		
		cornerSetRight := COMPLETE;			
		loadStepRight := COMPLETE;
		
END_CASE

//------------------------------------------------------------
IF cornerSetRight = COMPLETE THEN	
	loadStepRight := 0;
	cornerSetRight := 0;
	loadRightCornerCardboards := TRUE;
END_IF
END_METHOD

METHOD PROTECTED rightCornerSequence : BOOL
VAR_IN_OUT
	robot : RobotA22;
	skid : SkidMagazine;
	suctions : POINTER TO SuctionPad; //array of SuctionPads, casts from [1..3] to [0..2]
	loadStep : INT;
END_VAR
VAR_INPUT
	surfaceID : Surface;
	material : STRING;
	foldPos0 : INT;
	foldPos1 : INT;
END_VAR
VAR_OUTPUT
	error : BOOL;
END_VAR
VAR
	column : INT;
END_VAR
VAR CONSTANT
	suctionDistance : INT := 10;
END_VAR
{warning disable C0371}
IF material = '' THEN
	rightCornerSequence := TRUE;
	RETURN;
END_IF

CASE loadStep OF
	0:
		robot.clearCommand();
		IF robot.Ready THEN
			loadStep := 10;
		END_IF
		
	10: //overhead to insertion
		IF wrapper.Overhead = '' THEN
			RETURN;
		END_IF
		(*
		IF robot.eoatDistance < suctionDistance THEN
			robot.HoldMaterial := wrapper.Overhead;
		END_IF
		*)
	
		IF robot.Done THEN
			loadStep := COMPLETE;
			RETURN;
		END_IF
		
		CASE surfaceID OF
			Surface.TOP_RIGHT:		robot.setGroup(group := 1, value := A22.LOAD_OVERHEAD_TO_UPPER_CORNER);
			Surface.BOTTOM_RIGHT:	robot.setGroup(group := 1, value := A22.LOAD_OVERHEAD_TO_LOWER_CORNER);
		END_CASE
		robot.setGroup(group := 2, value := foldPos0);
		robot.setGroup(group := 3, value := foldPos1);
	
	COMPLETE:
		robot.clearCommand();
		
		CASE surfaceID OF
			Surface.TOP_RIGHT:		suctionTopRight[1].enable := suctionTopRight[3].enable := TRUE;
			Surface.BOTTOM_RIGHT:	suctionBottomRight[1].enable := suctionBottomRight[3].enable := TRUE;
		END_CASE
		
		//suctions[0].enable := TRUE;
		//suctions[2].enable := TRUE;
		
		rightCornerSequence := TRUE;
	
END_CASE
END_METHOD

END_FUNCTION_BLOCK

// ---- POUs/MAIN.TcPOU
PROGRAM MAIN
VAR_OUTPUT
	currentTime : TIMESTRUCT;
END_VAR
VAR
	execute : BOOL;
	manualStep : BOOL := TRUE;
	manualSuction : BOOL := FALSE;
	stop : BOOL;
	
	moduleA22 : CardboardCornerGuardEx;
END_VAR
VAR
	getLocalTime : FB_LocalSystemTime;
	test : BOOL;
END_VAR

CallHardwareModules(); //start program with hardware call

SetupHardware();

callModules();

CallHardwareModules(); //end program with hardware call

BundleJsonDemo();

ACTION callModules:
getLocalTime(
	sNetID:= '', 
	bEnable:= TRUE, 
	dwCycle:= , 
	dwOpt:= , 
	tTimeout:= , 
	bValid=> , 
	systemTime=> currentTime, 
	tzID=> );

moduleA22(
	execute:= execute, 
	stop:= stop, 
	manualStep:= manualStep, 
	manualSuction:= manualSuction, 
	
	benderLeft:= benderA22Left, 
	robotLeft:= robot3, 
	robotRight:= robot4, 
	skidLeft:= skidA22Left, 
	skidRight:= skidA22Right, 
	magazineLeft:= magazineA22Left, 
	magazineRight:= magazineA22Right, 
	wrapper:= wrapperA22, 
	horizontalDriveLeft:= horizontalDriveA22Left, 
	horizontalDriveRight:= horizontalDriveA22Right, 
	verticalDriveLeft:= verticalDriveA22Left, 
	verticalDriveRight:= verticalDriveA22Right, 
	pistonBottom:= pistonA22Bottom, 
	suctionTopLeft:= suctionA22TopLeft, 
	suctionTopRight:= suctionA22TopRight, 
	suctionBottomLeft:= suctionA22BottomLeft, 
	suctionBottomRight:= suctionA22BottomRight, 
	
	generalError=> , 
	failLeft=> , 
	failRight=> );
END_ACTION

END_PROGRAM

// ---- POUs/Hardware Calls/CallHardwareModules.TcPOU
FUNCTION CallHardwareModules : BOOL //only purpose of this function is to call modules from Hardware

robot3();
robot4();

skidA22Left(slots := skidSlotsA22Left, occupied := skidOccupancyA22Left, hmiTable := skidHmiA22Left);
skidA22Right(slots := skidSlotsA22Right, occupied := skidOccupancyA22Right, hmiTable := skidHmiA22Right);

magazineA22Left(slots := magazineSlotsA22Left, occupied := magazineOccupancyA22Left, hmiTable := magazineHmiA22Left);
magazineA22Right(slots := magazineSlotsA22Right, occupied := magazineOccupancyA22Right, hmiTable := magazineHmiA22Right);

wrapperA22();
benderA22Left();

horizontalDriveA22Left();
horizontalDriveA22Right();

verticalDriveA22Left();
verticalDriveA22Right();

pistonA22Bottom();

END_FUNCTION

// ---- POUs/Hardware Calls/SetupHardware.TcPOU
FUNCTION SetupHardware : BOOL
VAR
	iCardboardSlot : Cardboard;
	iCornerGuardSlot : CornerGuard;
	
	i : INT;
END_VAR

FOR iCardboardSlot:=1 TO Cardboard.size-1 BY 1 DO
	skidA22Left.setSlot(i := iCardboardSlot, material := TO_STRING(iCardboardSlot), error => );
	skidA22Right.setSlot(i := iCardboardSlot, material := TO_STRING(iCardboardSlot), error => );
END_FOR

//--------------------------------------------------

FOR iCornerGuardSlot:=1 TO CornerGuard.size-1 BY 1 DO
	magazineA22Left.setSlot(i := iCornerGuardSlot, material := TO_STRING(iCornerGuardSlot), error => );
	magazineA22Right.setSlot(i := iCornerGuardSlot, material := TO_STRING(iCornerGuardSlot), error => );
END_FOR

//--------------------------------------------------

FOR i:=1 TO GVL.maxQueue BY 1 DO
	{warning disable C0195}
	magazineA22Left.setOccupancy(i := i, occupancy := IntegerBitAccess( robot3.inputs[3], i-1) );
	skidA22Left.setOccupancy(i := i, occupancy := IntegerBitAccess( robot3.inputs[4], i-1) );
	
	magazineA22Right.setOccupancy(i := i, occupancy := IntegerBitAccess( robot4.inputs[3], i-1) );
	skidA22Right.setOccupancy(i := i, occupancy := IntegerBitAccess( robot4.inputs[4], i-1) );
	{warning restore C0195}
END_FOR

//--------------------------------------------------

verticalDriveA22Left.bEnable := 
verticalDriveA22Right.bEnable := 
horizontalDriveA22Left.bEnable := 
horizontalDriveA22Right.bEnable := 
pistonA22Bottom.bEnable := 
TRUE;

END_FUNCTION

// ---- POUs/Utility/IntegerBitAccess.TcPOU
FUNCTION IntegerBitAccess : BOOL
VAR_INPUT
	num : ANY_INT;
	n : ULINT;
END_VAR

IntegerBitAccess := (SHR(num, n) AND 1) > 0;

END_FUNCTION

// ---- POUs/BundleJsonDemo.TcPOU
PROGRAM BundleJsonDemo
VAR
	fbJson : FB_JsonSaxWriter;
	fbJsonDataType : FB_JsonReadWriteDataType;
	jsonDoc : STRING(100000); //this wont even show up in online view as twincat cannot show strings this long
	arrDoc : ARRAY[0..100000] OF BYTE;
	
	newBundle : Bundle;
	getBundle : Bundle;
END_VAR

newBundle.id := 'abcdefghijkl';
newBundle.autoRE := TRUE;
newBundle.cardboard := MAIN.moduleA22.materialsArr;
newBundle.timeDone := MAIN.currentTime;

fbJson.ResetDocument();
fbJsonDataType.AddJsonValueFromSymbol(fbJson, 'Bundle', SIZEOF(newBundle), ADR(newBundle));
fbJson.CopyDocument(jsonDoc, SIZEOF(jsonDoc));

MEMCPY(
	ADR(arrDoc), 
	ADR(jsonDoc),
	MIN(
		SIZEOF(jsonDoc),
		SIZEOF(arrDoc))
	);
	
fbJsonDataType.SetSymbolFromJson(jsonDoc, 'Bundle', SIZEOF(getBundle), ADR(getBundle));

END_PROGRAM

// ---- POUs/Hardware Calls/SuctionQuality.TcPOU
FUNCTION SuctionQuality : BOOL
VAR_IN_OUT
	suctions : ARRAY[*] OF SuctionPad;
END_VAR
VAR_INPUT
	insertionMaterial : STRING;
	recipeMaterial : STRING;
END_VAR
VAR
	i : DINT;
	
	failedVacuums : INT;
	numVacuums : INT;
END_VAR

(*
IF insertionMaterial <> recipeMaterial THEN //reintroduce this condition later
	RETURN;
END_IF
*)

FOR i:=LOWER_BOUND(suctions, 1) TO UPPER_BOUND(suctions, 1) BY 1 DO
	IF suctions[i].enable THEN
		numVacuums := numVacuums + 1;
		IF NOT suctions[i].occupied THEN
			failedVacuums := failedVacuums + 1;
		END_IF
	END_IF
	
END_FOR

SuctionQuality := TRUE;

END_FUNCTION

// ---- POUs/Utility/IntegerToBoolArray.TcPOU
FUNCTION IntegerToBoolArray : BOOL
VAR_IN_OUT
	arr : ARRAY[*] OF BOOL;
END_VAR
VAR_INPUT
	num : ANY_INT;
END_VAR
VAR_OUTPUT
	maxIterations : DINT;
END_VAR
VAR
	i : DINT;
	j : LINT;
END_VAR

maxIterations := MIN(
	(UPPER_BOUND(arr,1) - LOWER_BOUND(arr,1) + 1),
	num.diSize * 8);

FOR i:=LOWER_BOUND(arr, 1) TO UPPER_BOUND(arr, 1) BY 1 DO
	IF j < maxIterations THEN
		arr[i] := IntegerBitAccess(num, j);
		j := j + 1;
	END_IF
END_FOR

END_FUNCTION
